VAR_GLOBAL
	

	//MAIN/PACKML
	eCapPusherPackageState					:ARRAY [1..17] OF S_PackageState;		// [1..6] 

	(******P00_Alarms******)
	CapPusherGateError						:S_Error; 								// Szlaban
	CapPusherFeederError					:S_Error; 								// Podajnik
	CapPusherError							:S_Error;								// Wbijak

	(******P07_CapPusher********)	  

	//Szlaban
	bCapPusherGateRun						:BOOL;		

	//Podajnik
	bCapPusherFeederDoHoming				:BOOL;									// Wykonanie bazowania stacji podajnika 
	iCapPusherFeederTimeDelayOn				:INT; 										
	iCapPusherFeederTimeDelayOff			:INT; 
	iCapPusherFeederTimeToEmptySleeveError	:INT:=120;									// Czas do alarmu pustego rękawa 
	iCapPusherFeederCheckCountNOK			:INT;									// Zliczanie butelek bez nasadek

	//Zakrecanie
	bCapPusherDoHoming						:BOOL;									// Wykonanie bazowania stacji 
	bCapPusherEnable						:BOOL:=TRUE; 	
	iCapPusherTime							:INT; 	
	iCapPusherTime2							:INT;	

END_VAR

(*
VAR_GLOBAL PERSISTENT
	iRepairROPP1Counter						:INT;
	iRepairROPP2Counter						:INT;
	iRepairROPP3Counter						:INT;
	iRepairROPP4Counter						:INT;
END_VAR	*)

(* stored: Version 1.2.0.0, ProductVersion 3.1.4026.13, FileIdentifier b2d1e627a8d368dd73102bf15e037e6dd10c9102, FileSignature 08177a9e52865e18286be27cfc78a9c34fb5bff9f0b034e1bbc0ad1772dc3b456295e7905f62710cb5c97c75aefba0d834478365e1c339f7a4412071b80be9ab8d75d7609727f105c114fa39d96231ad7b90fac631afd29fcf1f7540dca53a30506f346c1a85971dbe768937d393898ca21e932716212f58bd19bbf7c1f5b081eaf3387a897751833ff3af892d453f35ef719ada19ae5a20f08d0967d700d2148961741b7b96264d455fb25d7c1656cba30688f49a81498e68a0b0a4cd64e4d4748b928e62312347ec643951958b1362d8e6783168c0d1474cf4b02e8dac7ae05af0e8261b967d3e3bdf2f4e26032510087a13394ea9715ff8a8b5e62e2b448b
   GVL GVL_CP: Id {c33b263d-fac9-4d0d-8598-a0065923d73b} *)
